PROGRAM P_Demo_FB_DMXSetDeviceLabel
VAR
    fbSetDeviceLabel  : FB_DMXSetDeviceLabel;         // 写设备标签
    stDmxCmdBuffer    : ST_DMXCommandBuffer;          // 与通讯 FB 共用
    wTargetManufId    : WORD := 16#4241;              // 目标灯具厂商 ID
    dwTargetDeviceId  : DWORD := 16#12131415;         // 目标灯具设备 ID
    byTargetPort      : BYTE := 0;                    // 根设备通道 0
    sNewLabel         : STRING := 'Stage-Left-Par-3'; // 要写入的设备名
    bDoSet            : BOOL := FALSE;                // 在线给一次上升沿触发
    bBusy             : BOOL;
    bError            : BOOL;
    udiErrId          : UDINT;
END_VAR

// ============================================================
// Tc2_DMX.FB_DMXSetDeviceLabel 演示程序
// ============================================================
// 场景：新装灯具调试时按布局给每盏灯写可读名字（如 Stage-Left-Par-3），写进设备本身。
// 价值：把命名信息固化到设备里，实现一次命名处处可读，比在各上位机各自维护映射表更可靠。
// 验证：设 sNewLabel，给 bDoSet 一次上升沿 -> bBusy 短暂 TRUE -> 回 FALSE 后用 FB_DMXGetDeviceLabel 回读应等于所写文本。
// 验证步骤：
//   1. 右键 PLC 项目下 POUs 文件夹 → Add → Existing Item → 选本 .TcPOU 文件
//   2. 引用 Tc2_DMX；同项目里放一个 FB_EL6851CommunicationEx 实例并共用 stDmxCmdBuffer（非 CycleMode）
//   3. 编译 → 登录 → 运行；按上方『验证』行在线给上升沿观察
// ============================================================

fbSetDeviceLabel(
    bStart                     := bDoSet,
    wDestinationManufacturerId := wTargetManufId,
    dwDestinationDeviceId      := dwTargetDeviceId,
    byPortId                   := byTargetPort,
    sDeviceLabel               := sNewLabel,
    dwOptions                  := 0,
    stCommandBuffer            := stDmxCmdBuffer,
    bBusy                      => bBusy,
    bError                     => bError,
    udiErrorId                 => udiErrId
);

END_PROGRAM

(* stored: Version 1.1.0.1, ProductVersion 3.1.4024.5
   POU P_Demo_FB_DMXSetDeviceLabel: Id {30f0139f-3cf4-5157-b611-714c896eac39}, SpecialFunc None *)
